# EPICS autosave request: BPMApp/Db/BPMRffe_settings.req
$(P)-$(BPM_NUMBER):RFFE:att1
$(P)-$(BPM_NUMBER):RFFE:att2
$(P)-$(BPM_NUMBER):RFFE:sw
